// Mitsubishi GX Works2 project: 演示程序   PLC: FX3U/FX3UC

PROGRAM MAIN
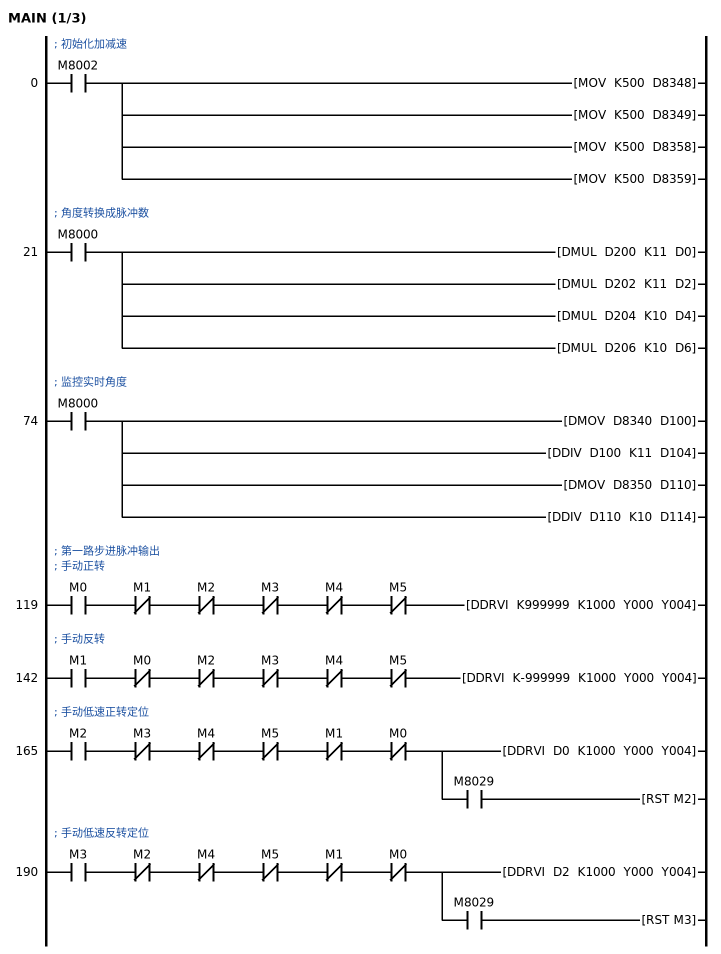
; 初始化加减速
0     LD      M8002
      MOV     K500 D8348
      MOV     K500 D8349
      MOV     K500 D8358
      MOV     K500 D8359
; 角度转换成脉冲数
21    LD      M8000
      DMUL    D200 K11 D0
      DMUL    D202 K11 D2
      DMUL    D204 K10 D4
      DMUL    D206 K10 D6
; 监控实时角度
74    LD      M8000
      DMOV    D8340 D100
      DDIV    D100 K11 D104
      DMOV    D8350 D110
      DDIV    D110 K10 D114
; 第一路步进脉冲输出
; 手动正转
119   LD      M0
      ANI     M1
      ANI     M2
      ANI     M3
      ANI     M4
      ANI     M5
      DDRVI   K999999 K1000 Y000 Y004
; 手动反转
142   LD      M1
      ANI     M0
      ANI     M2
      ANI     M3
      ANI     M4
      ANI     M5
      DDRVI   K-999999 K1000 Y000 Y004
; 手动低速正转定位
165   LD      M2
      ANI     M3
      ANI     M4
      ANI     M5
      ANI     M1
      ANI     M0
      DDRVI   D0 K1000 Y000 Y004
      AND     M8029
      RST     M2
; 手动低速反转定位
190   LD      M3
      ANI     M2
      ANI     M4
      ANI     M5
      ANI     M1
      ANI     M0
      DDRVI   D2 K1000 Y000 Y004
      AND     M8029
      RST     M3
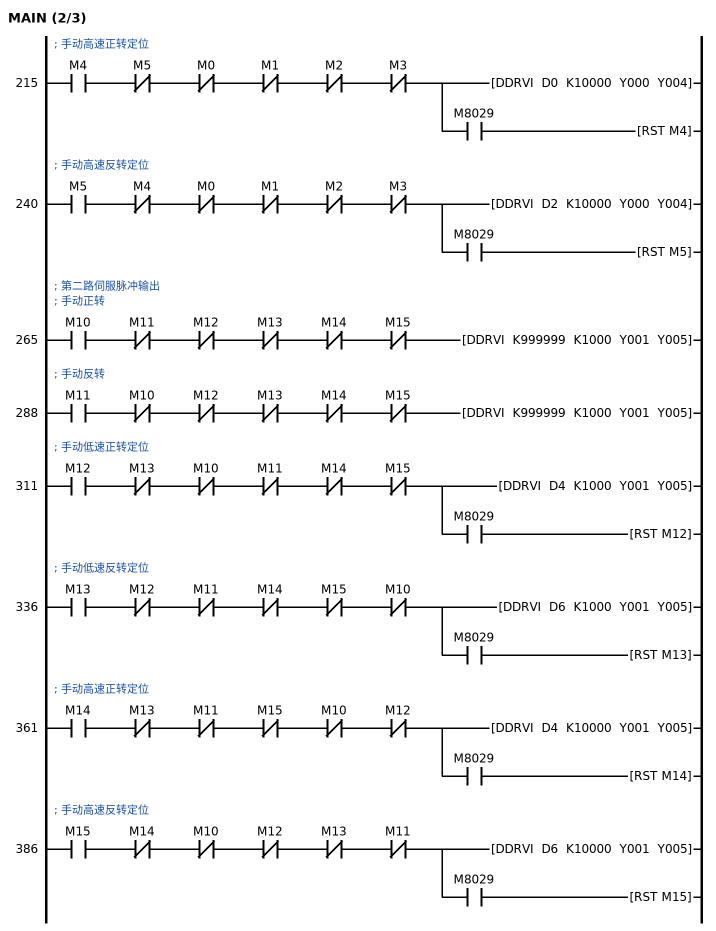
; 手动高速正转定位
215   LD      M4
      ANI     M5
      ANI     M0
      ANI     M1
      ANI     M2
      ANI     M3
      DDRVI   D0 K10000 Y000 Y004
      AND     M8029
      RST     M4
; 手动高速反转定位
240   LD      M5
      ANI     M4
      ANI     M0
      ANI     M1
      ANI     M2
      ANI     M3
      DDRVI   D2 K10000 Y000 Y004
      AND     M8029
      RST     M5
; 第二路伺服脉冲输出
; 手动正转
265   LD      M10
      ANI     M11
      ANI     M12
      ANI     M13
      ANI     M14
      ANI     M15
      DDRVI   K999999 K1000 Y001 Y005
; 手动反转
288   LD      M11
      ANI     M10
      ANI     M12
      ANI     M13
      ANI     M14
      ANI     M15
      DDRVI   K999999 K1000 Y001 Y005
; 手动低速正转定位
311   LD      M12
      ANI     M13
      ANI     M10
      ANI     M11
      ANI     M14
      ANI     M15
      DDRVI   D4 K1000 Y001 Y005
      AND     M8029
      RST     M12
; 手动低速反转定位
336   LD      M13
      ANI     M12
      ANI     M11
      ANI     M14
      ANI     M15
      ANI     M10
      DDRVI   D6 K1000 Y001 Y005
      AND     M8029
      RST     M13
; 手动高速正转定位
361   LD      M14
      ANI     M13
      ANI     M11
      ANI     M15
      ANI     M10
      ANI     M12
      DDRVI   D4 K10000 Y001 Y005
      AND     M8029
      RST     M14
; 手动高速反转定位
386   LD      M15
      ANI     M14
      ANI     M10
      ANI     M12
      ANI     M13
      ANI     M11
      DDRVI   D6 K10000 Y001 Y005
      AND     M8029
      RST     M15
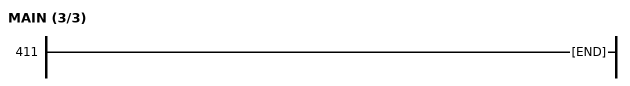
411   END
END_PROGRAM
